(* IEC 61131-3 sources: AXOpen/src/components.siemens.identification/ctrl/src/IOLink/AxoIOLinkRF200DataTypes, 14 files *)

(* ---- AxoIOLink_Header.st ---- *)
NAMESPACE AXOpen.Components.SIEM.Identification
    {S7.extern=ReadWrite}
    CLASS AxoIOLink_Header
        VAR PUBLIC
            call        :   AxoIOLink_HeaderCall;       //  header for read/write data record
            iolHeader   :   AxoIOLink_HeaderIolHeader;  //  header for IO-Link
        END_VAR
    END_CLASS
END_NAMESPACE

(* ---- AxoIOLink_HeaderCall.st ---- *)
NAMESPACE AXOpen.Components.SIEM.Identification
    {S7.extern=ReadWrite}
    CLASS AxoIOLink_HeaderCall
        VAR PUBLIC
            extFunctionNum  :	BYTE    :=  BYTE#16#08;     //  extended function number (fix coded 08h)
            port            :	BYTE    :=  BYTE#16#0;      //  variable port (user interface) 0...255
            fiIndex         :	WORD    :=  WORD#16#FE4A;   //	FI index (fix coded 65098)
        END_VAR
    END_CLASS
END_NAMESPACE

(* ---- AxoIOLink_HeaderIolHeader.st ---- *)
NAMESPACE AXOpen.Components.SIEM.Identification
    {S7.extern=ReadWrite}
    CLASS AxoIOLink_HeaderIolHeader
        VAR PUBLIC
            control         :	BYTE    :=  BYTE#16#0;  //  RD_WR = 0 = read = Control:=0x03 / / RD_WR = 1 = write = Control:=0x02
            indexHighByte   :	BYTE    :=  BYTE#16#0;  //  index of data record 0…32767 (high byte)
            indexLowByte    :	BYTE    :=  BYTE#16#0;  //  index of data record 0…32767 (low byte)
            subindex        :	BYTE    :=  BYTE#16#0;  //  subindex for data record 0...255
        END_VAR
    END_CLASS
END_NAMESPACE

(* ---- AxoIOLink_RF200_typeAll.st ---- *)
NAMESPACE AXOpen.Components.SIEM.Identification
    {S7.extern=ReadWrite}
    CLASS AxoIOLink_RF200_typeAll
        VAR PUBLIC
            directParameterPage     :	AxoIOLink_typeParameterPage0;       //  ID0: Parameter page 0
            systemCommand           :	BYTE    :=  BYTE#16#0;              //  ID2: System command
            deviceAccessLocks       :	WORD    :=  WORD#16#0;              //	ID12: Device access locks
            vendorName              :	STRING[12]  :=	'';                 //  ID16: Vendor name
            vendorText              :	STRING[12]  :=	'';                 //  ID17: Vendor text
            productName             :	STRING[24]  :=	'';                 //  ID18: Product name
            productID               :	STRING[16]  :=	'';                 //  ID19: Product ID
            productText             :	STRING[64]  :=	'';                 //  ID20: Product Text
            serialNumber            :	STRING[12]  :=	'';                 //  ID21: Serial Number
            hwRevision              :	STRING[12]  :=	'';                 //  ID22: Hardware revision
            fwRevision              :	STRING[12]  :=	'';                 //  ID23: Firmware revision
            appSpecificName         :	STRING[32]  :=	'';                 //  ID24: Application specific name
            errorCount              :	WORD    :=  WORD#16#0;              //	ID32: Number of errors that have occured (not warnings)
            deviceStatus            :	BYTE    :=  BYTE#16#0;              //  ID36: Device status
            deviceStatusDetailed    :	BYTE    :=  BYTE#16#0;              //  ID37: Detailed device status
            processImageIn          :	ARRAY[0..7] OF BYTE;                //	ID40: Read out last process image of the inputs
            processImageOut         :	ARRAY[0..7] OF BYTE;                //	ID41: Read out last process image of the outputs
            parameters              :	AxoIOLink_RF200_typeParameters;     //	ID64: Read/Write Reader Parameters
            eventHistory            :	AxoIOLink_RF200_typeEventHistory;   //	ID74: Number of events
            readerStatus            :	AxoIOLink_RF200_typeReaderStatus;   //	ID90: Reader status
            tagStatus               :	AxoIOLink_RF200_typeTagStatus;      //	ID91: Tag status
            uidHistory              :	AxoIOLink_RF200_typeUIDHistory;     //	ID92: History of UID
        END_VAR
    END_CLASS
END_NAMESPACE

(* ---- AxoIOLink_RF200_typeEventHistory.st ---- *)
NAMESPACE AXOpen.Components.SIEM.Identification
    {S7.extern=ReadWrite}
    CLASS AxoIOLink_RF200_typeEventHistory
        VAR PUBLIC
            lastEvent       :	DWORD   :=  DWORD#16#0; //  Last event
            secondLastEvent :	DWORD   :=  DWORD#16#0; //  Second last event
            thirdLastEvent  :	DWORD   :=  DWORD#16#0; //  Third last event
            fourthLastEvent :	DWORD   :=  DWORD#16#0; //  Fourth last event
            fifthLastEvent  :	DWORD   :=  DWORD#16#0; //  Fifth last event
        END_VAR
    END_CLASS
END_NAMESPACE

(* ---- AxoIOLink_RF200_typeParameters.st ---- *)
NAMESPACE AXOpen.Components.SIEM.Identification
    {S7.extern=ReadWrite}
    CLASS AxoIOLink_RF200_typeParameters
        VAR PUBLIC
            eventMessage    :	BYTE    :=  BYTE#16#0;  //  16#02: Event indication enabled (default), 16#04: No Message
            operatingMode   :	BYTE    :=  BYTE#16#0;  //  16#04: Scan UID (default), 16#08 Scan user data
            readyDelay      :	BYTE    :=  BYTE#16#0;  //  16#02 Turn off (default), 16#04: Turn on additional backup mechanism for
            dataHoldingTime :	BYTE    :=  BYTE#16#0;  //  Minimum time during which the process input data is not changed by the device
            rfParameters    :	BYTE    :=  BYTE#16#0;  //  Setting the RF parameters, 16#02 ISO default, 16#04: special settings
            modulation      :	BYTE    :=  BYTE#16#0;  //  Setting for the modulation strength 16#00 (0%) ... 16#64 (100%) - default 16#16 (22%)
            subcarrier      :	BYTE    :=  BYTE#16#0;  //  Subcarrier, 16#02: Single (default), 16#04: double
            dataTransfer    :	BYTE    :=  BYTE#16#0;  //  Data transmission speed, 16#02: low, 16#04: high (default)
        END_VAR
    END_CLASS
END_NAMESPACE

(* ---- AxoIOLink_RF200_typeReaderStatus.st ---- *)
NAMESPACE AXOpen.Components.SIEM.Identification
    {S7.extern=ReadWrite}
    CLASS AxoIOLink_RF200_typeReaderStatus
        VAR PUBLIC
            timeSinceStartup        :	DWORD   :=  DWORD#16#0; //  Operating time in seconds
            tagsInTheField          :	BYTE    :=  BYTE#16#0;  //  current number of transponders in the field
            antennaStatus           :	BYTE    :=  BYTE#16#0;  //  antenna turned on/off
            tagChanges              :	DWORD   :=  DWORD#16#0; //  number of transponder changes
            lineDriverRev           :	BYTE    :=  BYTE#16#0;  //  version of the IO-Link line driver
            errorCounterPassive     :	BYTE    :=  BYTE#16#0;  //  Air interface: Counter for errors in idle state
            abortCounter            :	BYTE    :=  BYTE#16#0;  //  Air interface: Communication aborted
            codeErrorCounter        :	BYTE    :=  BYTE#16#0;  //  Air interface: Communication disruption
            signatureErrorCounter   :	BYTE    :=  BYTE#16#0;  //  Air interface: Protocol error, signature error counter, is reset when read out
            crcErrorCounter         :	BYTE    :=  BYTE#16#0;  //  Air interface: Communication disruption
            currentCommandStatus    :	BYTE    :=  BYTE#16#0;  //  Command status of the last command, is reset when read out
            errorCount              :	BYTE    :=  BYTE#16#0;  //  HOST interface: Communication disruption
        END_VAR
    END_CLASS
END_NAMESPACE

(* ---- AxoIOLink_RF200_typeTagStatus.st ---- *)
NAMESPACE AXOpen.Components.SIEM.Identification
    {S7.extern=ReadWrite}
    CLASS AxoIOLink_RF200_typeTagStatus
        VAR PUBLIC
            uid             :	ARRAY[0..7] OF BYTE;	//  Unique identifier of the transponder
            tagName         :	BYTE    :=  BYTE#16#0;  //  Transponder Name
            chipVersion     :	BYTE    :=  BYTE#16#0;  //  Version of the Chip
            memSize         :	WORD    :=  WORD#16#0;  //  Memory size in Bytes
            lockStatus      :	BYTE    :=  BYTE#16#0;  //  Disable blocks on the chip
            memBlockSize    :	BYTE    :=  BYTE#16#0;  //  Size of memory blocks of the chip
            numBlocks       :	BYTE    :=  BYTE#16#0;  //  Number of memory blocks of the chip
        END_VAR
    END_CLASS
END_NAMESPACE

(* ---- AxoIOLink_RF200_typeUIDHistory.st ---- *)
NAMESPACE AXOpen.Components.SIEM.Identification
    {S7.extern=ReadWrite}
    CLASS AxoIOLink_RF200_typeUIDHistory
        VAR PUBLIC
            lastUID1        :  	DWORD   :=	DWORD#16#0; //  Last UID
            lastUID2        :  	DWORD   :=	DWORD#16#0; //  Last UID
            secondLastUID1  :	DWORD   :=	DWORD#16#0; //  Second last UID
            secondLastUID2  :	DWORD   :=	DWORD#16#0; //  Second last UID
            thirdLastUID1   :	DWORD   :=	DWORD#16#0; //  Third last UID
            thirdLastUID2   :	DWORD   :=	DWORD#16#0; //  Third last UID
            fourthLastUID1  :	DWORD   :=	DWORD#16#0; //  Fourth last UID
            fourthLastUID2  :	DWORD   :=	DWORD#16#0; //  Fourth last UID
            fifthLastUID1   :	DWORD   :=	DWORD#16#0; //  Fifth last UID
            fifthLastUID2   :	DWORD   :=	DWORD#16#0; //  Fifth last UID
        END_VAR
    END_CLASS
END_NAMESPACE

(* ---- AxoIOLink_RF200Device_Component_Status.st ---- *)
NAMESPACE AXOpen.Components.SIEM.Identification
    {S7.extern=ReadWrite}
    {#ix-attr:[Container(Layout.Stack)]}
    CLASS PUBLIC AxoIOLink_RF200Device_Component_Status  EXTENDS AXOpen.Components.Abstractions.AxoComponent_Status
        VAR PUBLIC
            Antenna_status      :   DWORD   :=  DWORD#16#0;
            ReadTag_status      :   DWORD   :=  DWORD#16#0;
            WriteTag_status     :   DWORD   :=  DWORD#16#0;
        END_VAR
    END_CLASS
END_NAMESPACE

(* ---- AxoIOLink_RF200Device_Config.st ---- *)
NAMESPACE AXOpen.Components.SIEM.Identification
    {S7.extern=ReadWrite}
    {#ix-attr:[Container(Layout.Stack)]}
    CLASS PUBLIC AxoIOLink_RF200Device_Config
        VAR PUBLIC
            {#ix-set:AttributeName = "<#Info time#>"}
            InfoTime : LTIME := LT#2S;
            {#ix-set:AttributeName = "<#Error time#>"}
            ErrorTime : LTIME := LT#5S;
        END_VAR
    END_CLASS
END_NAMESPACE

(* ---- AxoIOLink_RWdata.st ---- *)
NAMESPACE AXOpen.Components.SIEM.Identification
    {S7.extern=ReadWrite}
    CLASS AxoIOLink_RWdata
        VAR PUBLIC
            header  :   AxoIOLink_Header;       //  Header
            data    :   Array[0..231] OF BYTE;  //  Data
        END_VAR
    END_CLASS
END_NAMESPACE

(* ---- AxoIOLink_typeDiagnostics.st ---- *)
NAMESPACE AXOpen.Components.SIEM.Identification
    {S7.extern=ReadWrite}
    CLASS AxoIOLink_typeDiagnostics
        VAR PUBLIC
            status              :	WORD    :=  WORD#16#0;  //  Status of the Block or error identification when error occurred
            subfunctionStatus   :	DWORD   :=  DWORD#16#0; //  Status or return value of called FB's, FCs and system blocks
            stateNumber         :	DINT    :=  DINT#0;     //  State in the state machine of the block where the error occurred
        END_VAR
    END_CLASS
END_NAMESPACE

(* ---- AxoIOLink_typeParameterPage0.st ---- *)
NAMESPACE AXOpen.Components.SIEM.Identification
    {S7.extern=ReadWrite}
    CLASS AxoIOLink_typeParameterPage0
        VAR PUBLIC
            masterCommand       :	BYTE    :=  BYTE#16#00; // Switch the IO-Link operation mode (Fallback, Operate, Preoperate)
            masterCycleTime     :	BYTE    :=  BYTE#16#00; // Master Cycle Time
            minCycleTime        :	BYTE    :=  BYTE#16#00; // Minimum Device Cycle Time
            frameCapability     :	BYTE    :=  BYTE#16#00; // Supported frame types for communication
            ioLinkRevisionID    :	BYTE    :=  BYTE#16#00; // IO-Link protocol version implemented on the device
            processDataIn       :	BYTE    :=  BYTE#16#00; // Number and structure of the data process image of the inputs to the master
            processDataOut      :	BYTE    :=  BYTE#16#00; // Number and structure of the data process image of the outputs to the master
            vendorID1           :	BYTE    :=  BYTE#16#00; // Unique vendor identification number
            vendorID2           :	BYTE    :=  BYTE#16#00; // Siemens:0x002A
            deviceID1           :	BYTE    :=  BYTE#16#00; // Unique device identification number
            deviceID2           :	BYTE    :=  BYTE#16#00; // Unique device identification number
            deviceID3           :	BYTE    :=  BYTE#16#00; // Unique device identification number
            functionID1         :	BYTE    :=  BYTE#16#00; // Unique function identification number
            functionID2         :	BYTE    :=  BYTE#16#00; // Unique function identification number
            reserved1           :	BYTE    :=  BYTE#16#00; // Reserved
            reserved2           :	BYTE    :=  BYTE#16#00; // Reserved
        END_VAR
    END_CLASS
END_NAMESPACE
